TYPE E_ModalDesignationAbsInc :
(
	ModalDesignAbsInc_Undefined := 0,
	ModalDesignAbsInc_G90 := 4186,	//absolute designation
	ModalDesignAbsInc_G91 := 4187	//incremental designation
)UDINT;
END_TYPE

(* stored: Version 1.1.0.1, ProductVersion 3.1.0.25
   DUT E_ModalDesignationAbsInc: Id {4b9f64e2-adac-408c-9493-fc53021affd8} *)
